(* IEC 61131-3 sources: ArfBotOS/Codesys/Scripts/st, 4 files *)

(* ---- _00_Main_decl.st ---- *)
PROGRAM _00_Main
VAR
	//
    TaskInfo : POINTER TO CmpIecTask.Task_Info2;
    TaskHandle: CmpIecTask.RTS_IEC_HANDLE;
    Result: CmpIecTask.RTS_IEC_RESULT;

	// group handler for all motion fbs
	GroupHandler: FB_GroupHandler;

	// tuning
	MoveDistance: LREAL := 5.0;
	MoveRelative: ARRAY[0..5] OF MC_MoveRelative;
	EstimateDeadTime: ARRAY[0..5] OF SMC_EstimateDeadTime;
	TuneStart: ARRAY[0..5] OF BOOL;
	TraceStart: ARRAY[0..5] OF BOOL;
	TraceStop: ARRAY[0..5] OF BOOL;
	SetTuningMoveValues: BOOL:=TRUE;
	fCycleTimeMs: LREAL; (* MainTask / SoftMotion bus cycle, ms *)
	fMeasuredLagMs: ARRAY[0..5] OF LREAL;
	fEstimatedDeadTimeRaw: ARRAY[0..5] OF LREAL; (* unclamped SMC_EstimateDeadTime median *)
	fSuggestedDeadTime: ARRAY[0..5] OF LREAL; (* D in MainTask cycles, clamped to (0, 20] *)
	nDeadTimeSamples: ARRAY[0..5] OF INT;
	bDeadTimeSuggested: ARRAY[0..5] OF BOOL;
	UseSuggestedD: ARRAY[0..5] OF BOOL;
	sDeadTimeHelp: ARRAY[0..5] OF STRING(255);

	// homing
	ProcessHome: FB_HomingProcessor;
	HomingStatusText: STRING(255);

	// jogging
	ProcessJog: FB_JogProcessor;
	JogStatusText: STRING(255);
	ButtonTextIndex: INT:=0;

	// cnc
	VisuStruct3DControl_J: VisuStruct3DControl;
	TrackPosition: PositionTracker;

	// program processor
	ProcessPrograms: FB_ProgramProcessor;
	ProcessCommand_ActiveProgram: UINT := 0;
	ActiveCommandDetails: STRING(255):='';

	// controller
	Controller: FB_Controller;

	//
	EnableRtrig: R_TRIG;
	EnableFtrig: F_TRIG;
	_i, _j, _k: INT;
	BuildTests: BOOL:=FALSE;
	FirstScan: BOOL:=TRUE;

END_VAR

(* ---- _M_Tuning_decl.st ---- *)
METHOD PRIVATE _M_Tuning : BOOL
VAR_INPUT
END_VAR
VAR_STAT
	_MoveDelayTimer: ARRAY[0..5] OF TON;
	_TraceStartFtrig: ARRAY[0..5] OF F_TRIG;
	_MoveBusyFtrig: ARRAY[0..5] OF F_TRIG;
	_MoveBusyRtrig: ARRAY[0..5] OF R_TRIG;
	_MoveDelayTime: INT:=10; // ms
	_eDtState: ARRAY[0..5] OF INT; (* 0 idle, 1 wait cruise, 2 sampling, 3 done *)
	_bEstEnable: ARRAY[0..5] OF BOOL;
	_bDtFinish: ARRAY[0..5] OF BOOL;
	_aDtSample: ARRAY[0..5, 0..63] OF LREAL;
	_nSamples: ARRAY[0..5] OF INT;
	_fSetVel: LREAL;
	_fCruiseVel: LREAL;
	_fMedian: LREAL;
	_fSwap: LREAL;
	_fDtMin: LREAL := 0.1; (* SoftMotion rejects D = 0 *)
	_fDtMax: LREAL := 20.0; (* PosControl delay-buffer limit *)
	_fCruiseRatio: LREAL := 0.9;
	_nSampleMax: INT := 64;
	_i, _j, _k: INT;
END_VAR

(* ---- _M_Tuning_impl.st ---- *)
// MainTask interval is the SoftMotion bus cycle that D is counted in.
// TaskInfo.dwInterval is microseconds (simulation writes 1000).
IF GVL.dwMainInterval > 0 THEN
	fCycleTimeMs := DWORD_TO_LREAL(GVL.dwMainInterval) / 1000.0;
ELSE
	fCycleTimeMs := 1.0;
END_IF

IF FirstScan THEN
	FOR _i:=0 TO 5 BY 1 DO
		sDeadTimeHelp[_i] := 'SMC_EstimateDeadTime: START TUNE at Kp=0. Suggested D is the median of constant-velocity samples.';
	END_FOR
END_IF

// initial values
IF SetTuningMoveValues AND_THEN PersistentVars.Flags[GVL.INIT_DRV_IDX].Value THEN
	SetTuningMoveValues := FALSE;

	MoveRelative[0].Velocity := IoConfig_Globals.J1.fSWMaxVelocity;
	MoveRelative[0].Acceleration := IoConfig_Globals.J1.fSWMaxAcceleration;
	MoveRelative[0].Deceleration := IoConfig_Globals.J1.fSWMaxDeceleration;
	MoveRelative[0].Jerk := IoConfig_Globals.J1.fSWMaxJerk;
	MoveRelative[0].Distance := MoveDistance;

	MoveRelative[1].Velocity := IoConfig_Globals.J2.fSWMaxVelocity;
	MoveRelative[1].Acceleration := IoConfig_Globals.J2.fSWMaxAcceleration;
	MoveRelative[1].Deceleration := IoConfig_Globals.J2.fSWMaxDeceleration;
	MoveRelative[1].Jerk := IoConfig_Globals.J2.fSWMaxJerk;
	MoveRelative[1].Distance := MoveDistance;

	MoveRelative[2].Velocity := IoConfig_Globals.J3.fSWMaxVelocity;
	MoveRelative[2].Acceleration := IoConfig_Globals.J3.fSWMaxAcceleration;
	MoveRelative[2].Deceleration := IoConfig_Globals.J3.fSWMaxDeceleration;
	MoveRelative[2].Jerk := IoConfig_Globals.J3.fSWMaxJerk;
	MoveRelative[2].Distance := MoveDistance;

	MoveRelative[3].Velocity := IoConfig_Globals.J4.fSWMaxVelocity;
	MoveRelative[3].Acceleration := IoConfig_Globals.J4.fSWMaxAcceleration;
	MoveRelative[3].Deceleration := IoConfig_Globals.J4.fSWMaxDeceleration;
	MoveRelative[3].Jerk := IoConfig_Globals.J4.fSWMaxJerk;
	MoveRelative[3].Distance := MoveDistance;

	MoveRelative[4].Velocity := IoConfig_Globals.J5.fSWMaxVelocity;
	MoveRelative[4].Acceleration := IoConfig_Globals.J5.fSWMaxAcceleration;
	MoveRelative[4].Deceleration := IoConfig_Globals.J5.fSWMaxDeceleration;
	MoveRelative[4].Jerk := IoConfig_Globals.J5.fSWMaxJerk;
	MoveRelative[4].Distance := MoveDistance;

	MoveRelative[5].Velocity := IoConfig_Globals.J6.fSWMaxVelocity;
	MoveRelative[5].Acceleration := IoConfig_Globals.J6.fSWMaxAcceleration;
	MoveRelative[5].Deceleration := IoConfig_Globals.J6.fSWMaxDeceleration;
	MoveRelative[5].Jerk := IoConfig_Globals.J6.fSWMaxJerk;
	MoveRelative[5].Distance := MoveDistance;
END_IF

// trace activation
FOR _i:=0 TO 5 BY 1 DO

	IF TuneStart[_i] THEN
		TuneStart[_i] := FALSE;
		TraceStart[_i] := TRUE; // trace will handshake this bit low
		GroupHandler.M_EnableGroup();
		bDeadTimeSuggested[_i] := FALSE;
		fMeasuredLagMs[_i] := 0.0;
		fEstimatedDeadTimeRaw[_i] := 0.0;
		fSuggestedDeadTime[_i] := 0.0;
		nDeadTimeSamples[_i] := 0;
		_eDtState[_i] := 0;
		_bEstEnable[_i] := FALSE;
		_bDtFinish[_i] := FALSE;
		_nSamples[_i] := 0;
		sDeadTimeHelp[_i] := 'SMC_EstimateDeadTime: waiting for constant velocity. Kp=0 gives the cleanest estimate.';
	END_IF

	// copy a valid suggestion into the DeadTime spin; WRITE PARAMETERS still applies it
	IF UseSuggestedD[_i] THEN
		UseSuggestedD[_i] := FALSE;
		IF bDeadTimeSuggested[_i] THEN
			PersistentVars.PositionControllers[_i].fDeadTime := fSuggestedDeadTime[_i];
			sDeadTimeHelp[_i] := 'Copied suggested D into DeadTime. Press WRITE PARAMETERS to apply.';
		ELSE
			sDeadTimeHelp[_i] := 'No suggested D yet. Press START TUNE first.';
		END_IF
	END_IF

	// TraceStart will clear after handshake. this means the trace has started collecting samples
	// start the move delay timer to capture samples before the move
	_TraceStartFtrig[_i](CLK:=TraceStart[_i]);
	IF _TraceStartFtrig[_i].Q THEN
		_MoveDelayTimer[_i].IN:=TRUE;
	END_IF

	// once the move delay expires, start the move
	_MoveDelayTimer[_i](PT:=INT_TO_TIME(_MoveDelayTime));
	IF _MoveDelayTimer[_i].Q THEN
		_MoveDelayTimer[_i].IN:=FALSE;
		MoveRelative[_i].Execute := TRUE;
	END_IF

	_MoveBusyFtrig[_i](CLK:=MoveRelative[_i].Busy);
	IF _MoveBusyFtrig[_i].Q THEN
		MoveRelative[_i].Execute := FALSE;
		MoveRelative[_i].Distance := MoveRelative[_i].Distance * -1.0; // reverse direction
		_bEstEnable[_i] := FALSE;
		IF _eDtState[_i] = 2 THEN
			_bDtFinish[_i] := TRUE;
		ELSIF _eDtState[_i] = 1 THEN
			_eDtState[_i] := 0;
			sDeadTimeHelp[_i] := 'Move ended before constant velocity. Increase MoveDistance or reduce acceleration.';
		END_IF
	END_IF

	CASE _i OF
		0: _fSetVel := IoConfig_Globals.J1.fSetVelocity;
		1: _fSetVel := IoConfig_Globals.J2.fSetVelocity;
		2: _fSetVel := IoConfig_Globals.J3.fSetVelocity;
		3: _fSetVel := IoConfig_Globals.J4.fSetVelocity;
		4: _fSetVel := IoConfig_Globals.J5.fSetVelocity;
		5: _fSetVel := IoConfig_Globals.J6.fSetVelocity;
	END_CASE

	_MoveBusyRtrig[_i](CLK:=MoveRelative[_i].Busy);
	IF _MoveBusyRtrig[_i].Q THEN
		_nSamples[_i] := 0;
		nDeadTimeSamples[_i] := 0;
		_bDtFinish[_i] := FALSE;
		_eDtState[_i] := 1;
	END_IF

	_fCruiseVel := MoveRelative[_i].Velocity * _fCruiseRatio;
	IF _eDtState[_i] = 1 THEN
		IF ABS(_fSetVel) >= _fCruiseVel THEN
			_bEstEnable[_i] := TRUE;
			_eDtState[_i] := 2;
			sDeadTimeHelp[_i] := 'SMC_EstimateDeadTime: sampling at constant velocity...';
		END_IF
	END_IF

	IF _eDtState[_i] = 2 THEN
		IF _bEstEnable[_i] AND EstimateDeadTime[_i].Valid AND (_nSamples[_i] < _nSampleMax) THEN
			_aDtSample[_i, _nSamples[_i]] := ABS(EstimateDeadTime[_i].DeadTimeCycles);
			_nSamples[_i] := _nSamples[_i] + 1;
			nDeadTimeSamples[_i] := _nSamples[_i];
			IF _nSamples[_i] >= _nSampleMax THEN
				_bDtFinish[_i] := TRUE;
			END_IF
		END_IF
	END_IF

	IF _bDtFinish[_i] THEN
		_bDtFinish[_i] := FALSE;
		_bEstEnable[_i] := FALSE;
		_eDtState[_i] := 3;
		IF _nSamples[_i] < 1 THEN
			_eDtState[_i] := 0;
			sDeadTimeHelp[_i] := 'SMC_EstimateDeadTime never went Valid. Check enable and that the axis reached cruise.';
		ELSE
			// median of collected DeadTimeCycles
			FOR _j:=0 TO (_nSamples[_i] - 2) BY 1 DO
				FOR _k:=(_j + 1) TO (_nSamples[_i] - 1) BY 1 DO
					IF _aDtSample[_i, _k] < _aDtSample[_i, _j] THEN
						_fSwap := _aDtSample[_i, _j];
						_aDtSample[_i, _j] := _aDtSample[_i, _k];
						_aDtSample[_i, _k] := _fSwap;
					END_IF
				END_FOR
			END_FOR
			_fMedian := ABS(_aDtSample[_i, _nSamples[_i] / 2]);
			fEstimatedDeadTimeRaw[_i] := _fMedian;
			fMeasuredLagMs[_i] := _fMedian * fCycleTimeMs;
			IF _fMedian < _fDtMin THEN
				fSuggestedDeadTime[_i] := _fDtMin;
			ELSIF _fMedian > _fDtMax THEN
				fSuggestedDeadTime[_i] := _fDtMax;
			ELSE
				fSuggestedDeadTime[_i] := _fMedian;
			END_IF
			bDeadTimeSuggested[_i] := TRUE;
			sDeadTimeHelp[_i] := 'SMC_EstimateDeadTime median ';
			sDeadTimeHelp[_i] := CONCAT(sDeadTimeHelp[_i], TO_STRING(fEstimatedDeadTimeRaw[_i]));
			sDeadTimeHelp[_i] := CONCAT(sDeadTimeHelp[_i], ' cycles (');
			sDeadTimeHelp[_i] := CONCAT(sDeadTimeHelp[_i], TO_STRING(fMeasuredLagMs[_i]));
			sDeadTimeHelp[_i] := CONCAT(sDeadTimeHelp[_i], ' ms, n=');
			sDeadTimeHelp[_i] := CONCAT(sDeadTimeHelp[_i], INT_TO_STRING(_nSamples[_i]));
			IF fEstimatedDeadTimeRaw[_i] > _fDtMax THEN
				sDeadTimeHelp[_i] := CONCAT(sDeadTimeHelp[_i], '). Clamped to D 20 (PosControl max). WRITE PARAMETERS to apply.');
			ELSE
				sDeadTimeHelp[_i] := CONCAT(sDeadTimeHelp[_i], '). Suggested D ');
				sDeadTimeHelp[_i] := CONCAT(sDeadTimeHelp[_i], TO_STRING(fSuggestedDeadTime[_i]));
				sDeadTimeHelp[_i] := CONCAT(sDeadTimeHelp[_i], '. WRITE PARAMETERS to apply.');
			END_IF
		END_IF
	END_IF

END_FOR

// official SoftMotion estimator: enable only while at constant velocity
EstimateDeadTime[0](Axis:= IoConfig_Globals.J1, Enable:= _bEstEnable[0]);
EstimateDeadTime[1](Axis:= IoConfig_Globals.J2, Enable:= _bEstEnable[1]);
EstimateDeadTime[2](Axis:= IoConfig_Globals.J3, Enable:= _bEstEnable[2]);
EstimateDeadTime[3](Axis:= IoConfig_Globals.J4, Enable:= _bEstEnable[3]);
EstimateDeadTime[4](Axis:= IoConfig_Globals.J5, Enable:= _bEstEnable[4]);
EstimateDeadTime[5](Axis:= IoConfig_Globals.J6, Enable:= _bEstEnable[5]);

// move relative
MoveRelative[0](
	Axis:= IoConfig_Globals.J1,
	Execute:= ,
	Distance:= ,
	Velocity:= ,
	Acceleration:= ,
	Deceleration:= ,
	Jerk:= ,
	BufferMode:= ,
	Done=> ,
	Busy=> ,
	Active=> ,
	CommandAborted=> ,
	Error=> ,
	ErrorID=> );
MoveRelative[1](
	Axis:= IoConfig_Globals.J2,
	Execute:= ,
	Distance:= ,
	Velocity:= ,
	Acceleration:= ,
	Deceleration:= ,
	Jerk:= ,
	BufferMode:= ,
	Done=> ,
	Busy=> ,
	Active=> ,
	CommandAborted=> ,
	Error=> ,
	ErrorID=> );
MoveRelative[2](
	Axis:= IoConfig_Globals.J3,
	Execute:= ,
	Distance:= ,
	Velocity:= ,
	Acceleration:= ,
	Deceleration:= ,
	Jerk:= ,
	BufferMode:= ,
	Done=> ,
	Busy=> ,
	Active=> ,
	CommandAborted=> ,
	Error=> ,
	ErrorID=> );
MoveRelative[3](
	Axis:= IoConfig_Globals.J4,
	Execute:= ,
	Distance:= ,
	Velocity:= ,
	Acceleration:= ,
	Deceleration:= ,
	Jerk:= ,
	BufferMode:= ,
	Done=> ,
	Busy=> ,
	Active=> ,
	CommandAborted=> ,
	Error=> ,
	ErrorID=> );
MoveRelative[4](
	Axis:= IoConfig_Globals.J5,
	Execute:= ,
	Distance:= ,
	Velocity:= ,
	Acceleration:= ,
	Deceleration:= ,
	Jerk:= ,
	BufferMode:= ,
	Done=> ,
	Busy=> ,
	Active=> ,
	CommandAborted=> ,
	Error=> ,
	ErrorID=> );
MoveRelative[5](
	Axis:= IoConfig_Globals.J6,
	Execute:= ,
	Distance:= ,
	Velocity:= ,
	Acceleration:= ,
	Deceleration:= ,
	Jerk:= ,
	BufferMode:= ,
	Done=> ,
	Busy=> ,
	Active=> ,
	CommandAborted=> ,
	Error=> ,
	ErrorID=> );

(* ---- M_BuildTests_impl.st ---- *)
// taught positions referenced by factory programs
PersistentVars.StoredPositions[40].Position.X := -76.81;
PersistentVars.StoredPositions[40].Position.Y := 1.2;
PersistentVars.StoredPositions[40].Position.Z := -24.93;
PersistentVars.StoredPositions[40].Position.A := -4.74;
PersistentVars.StoredPositions[40].Position.B := 62.93;
PersistentVars.StoredPositions[40].Position.C := 24.21;
PersistentVars.StoredPositions[41].Comment := 'Euler Angle Tool Place Position MCS';
PersistentVars.StoredPositions[41].Position.X := 44.39;
PersistentVars.StoredPositions[41].Position.Y := -285.95;
PersistentVars.StoredPositions[41].Position.Z := 310.15;
PersistentVars.StoredPositions[41].Position.A := 96.6;
PersistentVars.StoredPositions[41].Position.B := 177.75;
PersistentVars.StoredPositions[41].Position.C := -174.21;
PersistentVars.StoredPositions[42].Comment := 'Euler Angle Tool Pick Position MCS';
PersistentVars.StoredPositions[42].Position.X := 43.97;
PersistentVars.StoredPositions[42].Position.Y := -280.38;
PersistentVars.StoredPositions[42].Position.Z := 215.24;
PersistentVars.StoredPositions[42].Position.A := 96.61;
PersistentVars.StoredPositions[42].Position.B := 177.75;
PersistentVars.StoredPositions[42].Position.C := -174.22;

//
FOR _i := GVL.PROG_CMDS_ARR_BEG TO GVL.PROG_CMDS_ARR_END BY 1 DO
	PersistentVars.Programs[0].Commands[_i].CommandType := DUT_CommandType.Disabled;
	PersistentVars.Programs[0].Commands[_i].CommandString := '';
	PersistentVars.Programs[0].Commands[_i].CommandComment := '';
END_FOR
PersistentVars.Programs[0].ProgramName := 'Pick and Place Euler Angle Tool';
PersistentVars.Programs[0].Commands[0].CommandType := DUT_CommandType.MoveCommand;
PersistentVars.Programs[0].Commands[0].CommandString := 'DIR ABS 50.0 ACS VAR STO 35 ';
PersistentVars.Programs[0].Commands[0].CommandComment := 'take on a pose';
PersistentVars.Programs[0].Commands[1].CommandType := DUT_CommandType.VarSetCommand;
PersistentVars.Programs[0].Commands[1].CommandString := 'STO 46 E 0.0 E 0.0 E 0.0 E 0.0 E 0.0 E 0.0 ';
PersistentVars.Programs[0].Commands[1].CommandComment := 'Rotate TCP according to ZYZ convention';
PersistentVars.Programs[0].Commands[3].CommandType := DUT_CommandType.LogicCommand;
PersistentVars.Programs[0].Commands[3].CommandString := 'IF REGISTER 40 EQU 0 THEN JUMP 5 ELSE JUMP 12 ';
PersistentVars.Programs[0].Commands[3].CommandComment := 'determine if pick or place';
PersistentVars.Programs[0].Commands[5].CommandType := DUT_CommandType.MoveCommand;
PersistentVars.Programs[0].Commands[5].CommandString := 'DIR ABS 50.0 MCS VAR STO 42 ';
PersistentVars.Programs[0].Commands[5].CommandComment := 'go to euler angle tool down position';
PersistentVars.Programs[0].Commands[6].CommandType := DUT_CommandType.OutputCommand;
PersistentVars.Programs[0].Commands[6].CommandString := 'DIG 0 1.0 ';
PersistentVars.Programs[0].Commands[6].CommandComment := 'open gripper';
PersistentVars.Programs[0].Commands[7].CommandType := DUT_CommandType.MoveCommand;
PersistentVars.Programs[0].Commands[7].CommandString := 'LIN REL 20.0 TCS LIT 0.0 0.0 25.0 0.0 0.0 0.0 ';
PersistentVars.Programs[0].Commands[7].CommandComment := 'move onto euler angle tool';
PersistentVars.Programs[0].Commands[8].CommandType := DUT_CommandType.OutputCommand;
PersistentVars.Programs[0].Commands[8].CommandString := 'DIG 0 0.0 ';
PersistentVars.Programs[0].Commands[8].CommandComment := 'close gripper';
PersistentVars.Programs[0].Commands[9].CommandType := DUT_CommandType.MoveCommand;
PersistentVars.Programs[0].Commands[9].CommandString := 'LIN REL 20.0 TCS LIT 0.0 0.0 -120.0 0.0 0.0 0.0 ';
PersistentVars.Programs[0].Commands[9].CommandComment := 'pull out tool';
PersistentVars.Programs[0].Commands[10].CommandType := DUT_CommandType.LogicCommand;
PersistentVars.Programs[0].Commands[10].CommandString := 'IF PASS THEN JUMP 16 ';
PersistentVars.Programs[0].Commands[12].CommandType := DUT_CommandType.MoveCommand;
PersistentVars.Programs[0].Commands[12].CommandString := 'DIR ABS 50.0 MCS VAR STO 41 ';
PersistentVars.Programs[0].Commands[12].CommandComment := 'go to euler angle tool up position';
PersistentVars.Programs[0].Commands[13].CommandType := DUT_CommandType.MoveCommand;
PersistentVars.Programs[0].Commands[13].CommandString := 'LIN REL 20.0 TCS LIT 0.0 0.0 120.0 0.0 0.0 0.0 ';
PersistentVars.Programs[0].Commands[13].CommandComment := 'push tool in';
PersistentVars.Programs[0].Commands[14].CommandType := DUT_CommandType.OutputCommand;
PersistentVars.Programs[0].Commands[14].CommandString := 'DIG 0 1.0 ';
PersistentVars.Programs[0].Commands[14].CommandComment := 'open gripper';
PersistentVars.Programs[0].Commands[15].CommandType := DUT_CommandType.MoveCommand;
PersistentVars.Programs[0].Commands[15].CommandString := 'LIN REL 20.0 TCS LIT 0.0 0.0 -25.0 0.0 0.0 0.0 ';
PersistentVars.Programs[0].Commands[15].CommandComment := 'move away from euler angle tool';

//
FOR _i := GVL.PROG_CMDS_ARR_BEG TO GVL.PROG_CMDS_ARR_END BY 1 DO
	PersistentVars.Programs[1].Commands[_i].CommandType := DUT_CommandType.Disabled;
	PersistentVars.Programs[1].Commands[_i].CommandString := '';
	PersistentVars.Programs[1].Commands[_i].CommandComment := '';
END_FOR
PersistentVars.Programs[1].ProgramName := 'Vision Pick and Place';
PersistentVars.Programs[1].Commands[0].CommandType := DUT_CommandType.VarSetCommand;
PersistentVars.Programs[1].Commands[0].CommandString := 'STO 46 E 0.0 E 0.0 E 0.0 E 0.0 E 0.0 E 90.0 ';
PersistentVars.Programs[1].Commands[0].CommandComment := 'Rotate TCP according to ZYZ convention';
PersistentVars.Programs[1].Commands[1].CommandType := DUT_CommandType.MoveCommand;
PersistentVars.Programs[1].Commands[1].CommandString := 'DIR ABS 60.0 ACS VAR STO 40 ';
PersistentVars.Programs[1].Commands[1].CommandComment := 'Take a pose';
PersistentVars.Programs[1].Commands[2].CommandType := DUT_CommandType.VisionCommand;
PersistentVars.Programs[1].Commands[2].CommandString := 'LOC 640 400 15 1 0.0 0.6 180.0 0 Pen.jpg FastTemplateMatching.py ';
PersistentVars.Programs[1].Commands[2].CommandComment := 'Find the object and store the result';
PersistentVars.Programs[1].Commands[3].CommandType := DUT_CommandType.VarSetCommand;
PersistentVars.Programs[1].Commands[3].CommandString := 'VIS 0 M -1.0 M -1.0 E -20.0 M -1.0 N 0.0 N 0.0 ';
PersistentVars.Programs[1].Commands[3].CommandComment := 'Rotate x and y to line up with TCP';
PersistentVars.Programs[1].Commands[4].CommandType := DUT_CommandType.MoveCommand;
PersistentVars.Programs[1].Commands[4].CommandString := 'DIR ABS 50.0 PC1 VAR VIS 0 ';
PersistentVars.Programs[1].Commands[4].CommandComment := 'Move over the object';
PersistentVars.Programs[1].Commands[5].CommandType := DUT_CommandType.OutputCommand;
PersistentVars.Programs[1].Commands[5].CommandString := 'DIG 0 1.0 ';
PersistentVars.Programs[1].Commands[5].CommandComment := 'Open the Gripper';
PersistentVars.Programs[1].Commands[6].CommandType := DUT_CommandType.MoveCommand;
PersistentVars.Programs[1].Commands[6].CommandString := 'LIN REL 50.0 TCS LIT 0.0 0.0 20.0 0.0 0.0 0.0 ';
PersistentVars.Programs[1].Commands[6].CommandComment := 'Move down to the object';
PersistentVars.Programs[1].Commands[7].CommandType := DUT_CommandType.OutputCommand;
PersistentVars.Programs[1].Commands[7].CommandString := 'DIG 0 0.0 ';
PersistentVars.Programs[1].Commands[7].CommandComment := 'Close the Gripper';
PersistentVars.Programs[1].Commands[8].CommandType := DUT_CommandType.PauseCommand;
PersistentVars.Programs[1].Commands[8].CommandString := 'T#1s';
PersistentVars.Programs[1].Commands[8].CommandComment := 'Pause while the gripper closes';
PersistentVars.Programs[1].Commands[9].CommandType := DUT_CommandType.MoveCommand;
PersistentVars.Programs[1].Commands[9].CommandString := 'LIN REL 50.0 TCS LIT 0.0 0.0 -20.0 0.0 0.0 0.0 ';
PersistentVars.Programs[1].Commands[9].CommandComment := 'Pick up the object';
PersistentVars.Programs[1].Commands[10].CommandType := DUT_CommandType.MoveCommand;
PersistentVars.Programs[1].Commands[10].CommandString := 'DIR ABS 50.0 PC1 LIT 0.0 0.0 -50.0 0.0 0.0 90.0 ';
PersistentVars.Programs[1].Commands[10].CommandComment := 'Move to drop position';
PersistentVars.Programs[1].Commands[11].CommandType := DUT_CommandType.OutputCommand;
PersistentVars.Programs[1].Commands[11].CommandString := 'DIG 0 1.0 ';
PersistentVars.Programs[1].Commands[11].CommandComment := 'Open the Gripper';

//
FOR _i := GVL.PROG_CMDS_ARR_BEG TO GVL.PROG_CMDS_ARR_END BY 1 DO
	PersistentVars.Programs[2].Commands[_i].CommandType := DUT_CommandType.Disabled;
	PersistentVars.Programs[2].Commands[_i].CommandString := '';
	PersistentVars.Programs[2].Commands[_i].CommandComment := '';
END_FOR
PersistentVars.Programs[2].ProgramName := 'PCS1 Corners';
PersistentVars.Programs[2].Commands[0].CommandType := DUT_CommandType.VarSetCommand;
PersistentVars.Programs[2].Commands[0].CommandString := 'STO 46 E 0.0 E 0.0 E 0.0 E 180.0 E 180.0 E 0.0 ';
PersistentVars.Programs[2].Commands[0].CommandComment := 'Rotate TCP according to ZYZ convention';
PersistentVars.Programs[2].Commands[1].CommandType := DUT_CommandType.VarSetCommand;
PersistentVars.Programs[2].Commands[1].CommandString := 'STO 48 E 282.23 E -0066.77 E 0195.00 E 0.0 E 0.0 E -0030.00 ';
PersistentVars.Programs[2].Commands[2].CommandType := DUT_CommandType.MoveCommand;
PersistentVars.Programs[2].Commands[2].CommandString := 'DIR ABS 050 PC1 LIT 0 0 0 0 0 0';
PersistentVars.Programs[2].Commands[3].CommandType := DUT_CommandType.MoveCommand;
PersistentVars.Programs[2].Commands[3].CommandString := 'LIN REL 100 TCS LIT 0.0 200.0 0.0 0.0 0.0 0.0';
PersistentVars.Programs[2].Commands[4].CommandType := DUT_CommandType.MoveCommand;
PersistentVars.Programs[2].Commands[4].CommandString := 'LIN REL 100 TCS LIT 00125.00 00000.00 00000.00 00000.00 00000.00 00000.00';
PersistentVars.Programs[2].Commands[5].CommandType := DUT_CommandType.MoveCommand;
PersistentVars.Programs[2].Commands[5].CommandString := 'LIN REL 100 TCS LIT 00000.00 -0200.00 00000.00 00000.00 00000.00 00000.00';
PersistentVars.Programs[2].Commands[6].CommandType := DUT_CommandType.MoveCommand;
PersistentVars.Programs[2].Commands[6].CommandString := 'LIN REL 100 TCS LIT -0125.00 00000.00 00000.00 00000.00 00000.00 00000.00';
PersistentVars.Programs[2].Commands[7].CommandType := DUT_CommandType.MoveCommand;
PersistentVars.Programs[2].Commands[7].CommandString := 'DIR ABS 050 ACS LIT +00 +30 -30 +00 +30 +00';

//
FOR _i := GVL.PROG_CMDS_ARR_BEG TO GVL.PROG_CMDS_ARR_END BY 1 DO
	PersistentVars.Programs[3].Commands[_i].CommandType := DUT_CommandType.Disabled;
	PersistentVars.Programs[3].Commands[_i].CommandString := '';
	PersistentVars.Programs[3].Commands[_i].CommandComment := '';
END_FOR
PersistentVars.Programs[3].ProgramName := 'Cnc Validation';
PersistentVars.Programs[3].Commands[0].CommandType := DUT_CommandType.VarSetCommand;
PersistentVars.Programs[3].Commands[0].CommandString := 'STO 46 E 0.0 E 0.0 E 0.0 E 0.0 E 0.0 E 0.0 ';
PersistentVars.Programs[3].Commands[0].CommandComment := 'Clear TCP Offset';
PersistentVars.Programs[3].Commands[2].CommandType := DUT_CommandType.MoveCommand;
PersistentVars.Programs[3].Commands[2].CommandString := 'DIR ABS 50.0 ACS VAR STO 37 ';
PersistentVars.Programs[3].Commands[2].CommandComment := 'Move to Pose 4';
PersistentVars.Programs[3].Commands[3].CommandType := DUT_CommandType.CncCommand;
PersistentVars.Programs[3].Commands[3].CommandString := 'CNC_Cone.cnc ';
PersistentVars.Programs[3].Commands[3].CommandComment := 'Run the cnc file on disk';
PersistentVars.Programs[3].Commands[5].CommandType := DUT_CommandType.MoveCommand;
PersistentVars.Programs[3].Commands[5].CommandString := 'DIR ABS 50.0 ACS VAR STO 34 ';
PersistentVars.Programs[3].Commands[5].CommandComment := 'Move to Pose 1';
PersistentVars.Programs[3].Commands[6].CommandType := DUT_CommandType.CncCommand;
PersistentVars.Programs[3].Commands[6].CommandString := 'CNC_FromFile.cnc ';
PersistentVars.Programs[3].Commands[6].CommandComment := 'Run the cnc file on disk';

//
FOR _i := GVL.PROG_CMDS_ARR_BEG TO GVL.PROG_CMDS_ARR_END BY 1 DO
	PersistentVars.Programs[4].Commands[_i].CommandType := DUT_CommandType.Disabled;
	PersistentVars.Programs[4].Commands[_i].CommandString := '';
	PersistentVars.Programs[4].Commands[_i].CommandComment := '';
END_FOR
PersistentVars.Programs[4].ProgramName := 'Vision Validation';
PersistentVars.Programs[4].Commands[0].CommandType := DUT_CommandType.VisionCommand;
PersistentVars.Programs[4].Commands[0].CommandString := 'CAL 640 400 60 22.0 6 9 ';
PersistentVars.Programs[4].Commands[0].CommandComment := 'Calibrate using checkerboard';
PersistentVars.Programs[4].Commands[2].CommandType := DUT_CommandType.PauseCommand;
PersistentVars.Programs[4].Commands[2].CommandString := 'T#10s ';
PersistentVars.Programs[4].Commands[2].CommandComment := 'Wait 10 seconds';
PersistentVars.Programs[4].Commands[4].CommandType := DUT_CommandType.VisionCommand;
PersistentVars.Programs[4].Commands[4].CommandString := 'LOC 640 400 60 1 0.0 0.8 30.0 10 Template.jpg FastTemplateMatching.py';
PersistentVars.Programs[4].Commands[4].CommandComment := 'Find the template';

//
FOR _i := GVL.PROG_CMDS_ARR_BEG TO GVL.PROG_CMDS_ARR_END BY 1 DO
	PersistentVars.Programs[5].Commands[_i].CommandType := DUT_CommandType.Disabled;
	PersistentVars.Programs[5].Commands[_i].CommandString := '';
	PersistentVars.Programs[5].Commands[_i].CommandComment := '';
END_FOR
PersistentVars.Programs[5].ProgramName := 'VarSet Validation';
PersistentVars.Programs[5].Commands[0].CommandType := DUT_CommandType.VarSetCommand;
PersistentVars.Programs[5].Commands[0].CommandString := 'STO 1 E 6.0 E 5.0 E 4.0 E 3.0 E 2.0 E 1.0 ';
PersistentVars.Programs[5].Commands[1].CommandType := DUT_CommandType.VarSetCommand;
PersistentVars.Programs[5].Commands[1].CommandString := 'VIS 2 1 2 3 4 5 6';
PersistentVars.Programs[5].Commands[2].CommandType := DUT_CommandType.VarSetCommand;
PersistentVars.Programs[5].Commands[2].CommandString := 'FLG 3 1';

//
FOR _i := GVL.PROG_CMDS_ARR_BEG TO GVL.PROG_CMDS_ARR_END BY 1 DO
	PersistentVars.Programs[6].Commands[_i].CommandType := DUT_CommandType.Disabled;
	PersistentVars.Programs[6].Commands[_i].CommandString := '';
	PersistentVars.Programs[6].Commands[_i].CommandComment := '';
END_FOR
PersistentVars.Programs[6].ProgramName := 'Logic Validation';
PersistentVars.Programs[6].Commands[0].CommandType := DUT_CommandType.LogicCommand;
PersistentVars.Programs[6].Commands[0].CommandString := 'IF INPUT 1 EQU 1 THEN OUTPUT 1 1 ELSE OUTPUT 1 0';
PersistentVars.Programs[6].Commands[1].CommandType := DUT_CommandType.LogicCommand;
PersistentVars.Programs[6].Commands[1].CommandString := 'IF INPUT 1 EQU 1 THEN CNTUP 1 ELSE CNTUP 2';
PersistentVars.Programs[6].Commands[2].CommandType := DUT_CommandType.LogicCommand;
PersistentVars.Programs[6].Commands[2].CommandString := 'IF COUNTER 2 GRE 10 THEN NOP ELSE JUMP 0';

//
FOR _i := GVL.PROG_CMDS_ARR_BEG TO GVL.PROG_CMDS_ARR_END BY 1 DO
	PersistentVars.Programs[7].Commands[_i].CommandType := DUT_CommandType.Disabled;
	PersistentVars.Programs[7].Commands[_i].CommandString := '';
	PersistentVars.Programs[7].Commands[_i].CommandComment := '';
END_FOR
PersistentVars.Programs[7].ProgramName := 'Euler Angles Demo';
PersistentVars.Programs[7].Commands[0].CommandType := DUT_CommandType.LogicCommand;
PersistentVars.Programs[7].Commands[0].CommandString := 'IF PASS THEN REGISTER 40 0 ';
PersistentVars.Programs[7].Commands[0].CommandComment := 'Set pick/place register to pick tool';
PersistentVars.Programs[7].Commands[1].CommandType := DUT_CommandType.LogicCommand;
PersistentVars.Programs[7].Commands[1].CommandString := 'IF PASS THEN CALL 0 ';
PersistentVars.Programs[7].Commands[1].CommandComment := 'Call pick and place program';
PersistentVars.Programs[7].Commands[3].CommandType := DUT_CommandType.LogicCommand;
PersistentVars.Programs[7].Commands[3].CommandString := 'IF COUNTER 7 EQU 0 THEN NOP ELSE JUMP 7 ';
PersistentVars.Programs[7].Commands[3].CommandComment := 'apply or jump over';
PersistentVars.Programs[7].Commands[4].CommandType := DUT_CommandType.VarSetCommand;
PersistentVars.Programs[7].Commands[4].CommandString := 'STO 46 E 0.0 E 0.0 E 70.0 E 0.0 E 0.0 E 0.0 ';
PersistentVars.Programs[7].Commands[4].CommandComment := 'offset TCP Z';
PersistentVars.Programs[7].Commands[5].CommandType := DUT_CommandType.LogicCommand;
PersistentVars.Programs[7].Commands[5].CommandString := 'IF PASS THEN JUMP 19 ';
PersistentVars.Programs[7].Commands[5].CommandComment := 'go to move commands';
PersistentVars.Programs[7].Commands[7].CommandType := DUT_CommandType.LogicCommand;
PersistentVars.Programs[7].Commands[7].CommandString := 'IF COUNTER 7 EQU 1 THEN NOP ELSE JUMP 11 ';
PersistentVars.Programs[7].Commands[7].CommandComment := 'apply or jump over';
PersistentVars.Programs[7].Commands[8].CommandType := DUT_CommandType.VarSetCommand;
PersistentVars.Programs[7].Commands[8].CommandString := 'STO 46 E 0.0 E 0.0 E 170.0 E 0.0 E 0.0 E 0.0 ';
PersistentVars.Programs[7].Commands[8].CommandComment := 'offset TCP Z';
PersistentVars.Programs[7].Commands[9].CommandType := DUT_CommandType.LogicCommand;
PersistentVars.Programs[7].Commands[9].CommandString := 'IF PASS THEN JUMP 19 ';
PersistentVars.Programs[7].Commands[9].CommandComment := 'go to move commands';
PersistentVars.Programs[7].Commands[11].CommandType := DUT_CommandType.LogicCommand;
PersistentVars.Programs[7].Commands[11].CommandString := 'IF COUNTER 7 EQU 2 THEN NOP ELSE JUMP 15 ';
PersistentVars.Programs[7].Commands[11].CommandComment := 'apply or jump over';
PersistentVars.Programs[7].Commands[12].CommandType := DUT_CommandType.VarSetCommand;
PersistentVars.Programs[7].Commands[12].CommandString := 'STO 46 E 0.0 E -100.0 E 70.0 E 0.0 E 0.0 E 0.0 ';
PersistentVars.Programs[7].Commands[12].CommandComment := 'offset TCP X and Y';
PersistentVars.Programs[7].Commands[13].CommandType := DUT_CommandType.LogicCommand;
PersistentVars.Programs[7].Commands[13].CommandString := 'IF PASS THEN JUMP 19 ';
PersistentVars.Programs[7].Commands[13].CommandComment := 'go to move commands';
PersistentVars.Programs[7].Commands[15].CommandType := DUT_CommandType.LogicCommand;
PersistentVars.Programs[7].Commands[15].CommandString := 'IF COUNTER 7 EQU 3 THEN NOP ELSE JUMP 29 ';
PersistentVars.Programs[7].Commands[15].CommandComment := 'apply or jump over';
PersistentVars.Programs[7].Commands[16].CommandType := DUT_CommandType.VarSetCommand;
PersistentVars.Programs[7].Commands[16].CommandString := 'STO 46 E 100.0 E 0.0 E 70.0 E 0.0 E 0.0 E 0.0 ';
PersistentVars.Programs[7].Commands[16].CommandComment := 'offset TCP X and Z';
PersistentVars.Programs[7].Commands[17].CommandType := DUT_CommandType.LogicCommand;
PersistentVars.Programs[7].Commands[17].CommandString := 'IF PASS THEN JUMP 19 ';
PersistentVars.Programs[7].Commands[17].CommandComment := 'go to move commands';
PersistentVars.Programs[7].Commands[19].CommandType := DUT_CommandType.MoveCommand;
PersistentVars.Programs[7].Commands[19].CommandString := 'DIR ABS 50.0 ACS VAR STO 35 ';
PersistentVars.Programs[7].Commands[19].CommandComment := 'take on a pose';
PersistentVars.Programs[7].Commands[20].CommandType := DUT_CommandType.MoveCommand;
PersistentVars.Programs[7].Commands[20].CommandString := 'LIN ABS 70.0 TCS LIT 0.0 0.0 0.0 0.0 0.0 -45.0 ';
PersistentVars.Programs[7].Commands[20].CommandComment := 'rotate TCP Z with ZYZ convention';
PersistentVars.Programs[7].Commands[21].CommandType := DUT_CommandType.MoveCommand;
PersistentVars.Programs[7].Commands[21].CommandString := 'LIN ABS 70.0 TCS LIT 0.0 0.0 0.0 0.0 -30.0 0.0 ';
PersistentVars.Programs[7].Commands[21].CommandComment := 'rotate around TCP Y with ZYZ convention';
PersistentVars.Programs[7].Commands[22].CommandType := DUT_CommandType.MoveCommand;
PersistentVars.Programs[7].Commands[22].CommandString := 'LIN ABS 70.0 TCS LIT 0.0 0.0 0.0 90.0 30.0 -90.0 ';
PersistentVars.Programs[7].Commands[22].CommandComment := 'rotate around TCP X with ZYZ convention';
PersistentVars.Programs[7].Commands[23].CommandType := DUT_CommandType.MoveCommand;
PersistentVars.Programs[7].Commands[23].CommandString := 'LIN ABS 70.0 TCS LIT 0.0 0.0 0.0 90.0 -30.0 -90.0 ';
PersistentVars.Programs[7].Commands[23].CommandComment := 'rotate around TCP X with ZYZ convention';
PersistentVars.Programs[7].Commands[24].CommandType := DUT_CommandType.MoveCommand;
PersistentVars.Programs[7].Commands[24].CommandString := 'LIN ABS 70.0 TCS LIT 0.0 0.0 0.0 0.0 30.0 0.0 ';
PersistentVars.Programs[7].Commands[24].CommandComment := 'rotate around TCP Y with ZYZ convention';
PersistentVars.Programs[7].Commands[25].CommandType := DUT_CommandType.MoveCommand;
PersistentVars.Programs[7].Commands[25].CommandString := 'DIR ABS 70.0 ACS VAR STO 35 ';
PersistentVars.Programs[7].Commands[25].CommandComment := 'take on a pose';
PersistentVars.Programs[7].Commands[27].CommandType := DUT_CommandType.LogicCommand;
PersistentVars.Programs[7].Commands[27].CommandString := 'IF PASS THEN CNTUP 7 ';
PersistentVars.Programs[7].Commands[27].CommandComment := 'count up counter';
PersistentVars.Programs[7].Commands[28].CommandType := DUT_CommandType.LogicCommand;
PersistentVars.Programs[7].Commands[28].CommandString := 'IF PASS THEN JUMP 3 ';
PersistentVars.Programs[7].Commands[28].CommandComment := 'go back to start';
PersistentVars.Programs[7].Commands[29].CommandType := DUT_CommandType.LogicCommand;
PersistentVars.Programs[7].Commands[29].CommandString := 'IF PASS THEN CNTRST 7 ';
PersistentVars.Programs[7].Commands[29].CommandComment := 'reset counter back to 0';
PersistentVars.Programs[7].Commands[31].CommandType := DUT_CommandType.LogicCommand;
PersistentVars.Programs[7].Commands[31].CommandString := 'IF PASS THEN REGISTER 40 1 ';
PersistentVars.Programs[7].Commands[31].CommandComment := 'Set pick/place register to place tool';
PersistentVars.Programs[7].Commands[32].CommandType := DUT_CommandType.LogicCommand;
PersistentVars.Programs[7].Commands[32].CommandString := 'IF PASS THEN CALL 0 ';
PersistentVars.Programs[7].Commands[32].CommandComment := 'Call pick and place program';

//
FOR _i := GVL.PROG_CMDS_ARR_BEG TO GVL.PROG_CMDS_ARR_END BY 1 DO
	PersistentVars.Programs[9].Commands[_i].CommandType := DUT_CommandType.Disabled;
	PersistentVars.Programs[9].Commands[_i].CommandString := '';
	PersistentVars.Programs[9].Commands[_i].CommandComment := '';
END_FOR
PersistentVars.Programs[9].ProgramName := 'Vision PCS1 Test';
PersistentVars.Programs[9].Commands[0].CommandType := DUT_CommandType.MoveCommand;
PersistentVars.Programs[9].Commands[0].CommandString := 'DIR ABS 75.0 ACS VAR STO 35 ';
PersistentVars.Programs[9].Commands[0].CommandComment := 'Move to Pose 2';
PersistentVars.Programs[9].Commands[2].CommandType := DUT_CommandType.VarSetCommand;
PersistentVars.Programs[9].Commands[2].CommandString := 'STO 48 E 241.75 E -54.39 E 203.17 E 0.0 E 181.0 E -90.0 ';
PersistentVars.Programs[9].Commands[2].CommandComment := 'Set PCS1 Offset in ZYZ';
PersistentVars.Programs[9].Commands[3].CommandType := DUT_CommandType.VarSetCommand;
PersistentVars.Programs[9].Commands[3].CommandString := 'STO 46 E 0.0 E 0.0 E 0.0 E 0.0 E 0.0 E 90.0 ';
PersistentVars.Programs[9].Commands[3].CommandComment := 'Rotate TCP in ZYZ';
PersistentVars.Programs[9].Commands[5].CommandType := DUT_CommandType.VisionCommand;
PersistentVars.Programs[9].Commands[5].CommandString := 'LOC 640 400 15 2 0.0 0.8 180.0 0 screwdriver1.jpg FastTemplateMatching.py ';
PersistentVars.Programs[9].Commands[5].CommandComment := 'Find the object and store the result';
PersistentVars.Programs[9].Commands[7].CommandType := DUT_CommandType.LogicCommand;
PersistentVars.Programs[9].Commands[7].CommandString := 'IF REGISTER 0 EQU 0 THEN JUMP 14 ELSE NOP ';
PersistentVars.Programs[9].Commands[7].CommandComment := 'If parts count = 0 jump to end';
PersistentVars.Programs[9].Commands[9].CommandType := DUT_CommandType.MoveCommand;
PersistentVars.Programs[9].Commands[9].CommandString := 'DIR ABS 50.0 PC1 VAR VIS 0 ';
PersistentVars.Programs[9].Commands[9].CommandComment := 'Move over the object';
PersistentVars.Programs[9].Commands[10].CommandType := DUT_CommandType.PauseCommand;
PersistentVars.Programs[9].Commands[10].CommandString := 'T#3s ';
PersistentVars.Programs[9].Commands[12].CommandType := DUT_CommandType.LogicCommand;
PersistentVars.Programs[9].Commands[12].CommandString := 'IF REGISTER 0 GRT 1 THEN JUMP 0 ELSE NOP ';
PersistentVars.Programs[9].Commands[12].CommandComment := 'If more than 1 part go again';
PersistentVars.Programs[9].Commands[14].CommandType := DUT_CommandType.MoveCommand;
PersistentVars.Programs[9].Commands[14].CommandString := 'DIR ABS 75.0 ACS VAR STO 35 ';
PersistentVars.Programs[9].Commands[14].CommandComment := 'Move to Pose 2';

//
FOR _i := GVL.PROG_CMDS_ARR_BEG TO GVL.PROG_CMDS_ARR_END BY 1 DO
	PersistentVars.Programs[10].Commands[_i].CommandType := DUT_CommandType.Disabled;
	PersistentVars.Programs[10].Commands[_i].CommandString := '';
	PersistentVars.Programs[10].Commands[_i].CommandComment := '';
END_FOR
PersistentVars.Programs[10].ProgramName := 'Pick Glow Stick';
PersistentVars.Programs[10].Commands[0].CommandType := DUT_CommandType.LogicCommand;
PersistentVars.Programs[10].Commands[0].CommandString := 'IF REGISTER 2 EQU 0 THEN NOP ELSE JUMP 5 ';
PersistentVars.Programs[10].Commands[0].CommandComment := 'check if initialized';
PersistentVars.Programs[10].Commands[1].CommandType := DUT_CommandType.VarSetCommand;
PersistentVars.Programs[10].Commands[1].CommandString := 'STO 0 E 0.0 E 0.0 E 0.0 E 0.0 E 0.0 E 0.0 ';
PersistentVars.Programs[10].Commands[1].CommandComment := 'clear out the tcp position';
PersistentVars.Programs[10].Commands[2].CommandType := DUT_CommandType.LogicCommand;
PersistentVars.Programs[10].Commands[2].CommandString := 'IF PASS THEN CNTRST 0 ';
PersistentVars.Programs[10].Commands[2].CommandComment := 'clear column counter';
PersistentVars.Programs[10].Commands[3].CommandType := DUT_CommandType.LogicCommand;
PersistentVars.Programs[10].Commands[3].CommandString := 'IF PASS THEN CNTRST 1 ';
PersistentVars.Programs[10].Commands[3].CommandComment := 'clear row counter';
PersistentVars.Programs[10].Commands[4].CommandType := DUT_CommandType.LogicCommand;
PersistentVars.Programs[10].Commands[4].CommandString := 'IF PASS THEN REGISTER 2 1 ';
PersistentVars.Programs[10].Commands[4].CommandComment := 'mark data initialized';
PersistentVars.Programs[10].Commands[6].CommandType := DUT_CommandType.MoveCommand;
PersistentVars.Programs[10].Commands[6].CommandString := 'DIR ABS 50.0 ACS VAR STO 34 ';
PersistentVars.Programs[10].Commands[6].CommandComment := 'take on a pose';
PersistentVars.Programs[10].Commands[7].CommandType := DUT_CommandType.OutputCommand;
PersistentVars.Programs[10].Commands[7].CommandString := 'DIG 0 1.0 ';
PersistentVars.Programs[10].Commands[7].CommandComment := 'open gripper';
PersistentVars.Programs[10].Commands[8].CommandType := DUT_CommandType.MoveCommand;
PersistentVars.Programs[10].Commands[8].CommandString := 'LIN ABS 50.0 PC1 VAR STO 0 ';
PersistentVars.Programs[10].Commands[8].CommandComment := 'go to the pick position in PCS1';
PersistentVars.Programs[10].Commands[9].CommandType := DUT_CommandType.MoveCommand;
PersistentVars.Programs[10].Commands[9].CommandString := 'LIN REL 50.0 TCS LIT 0.0 0.0 10.0 0.0 0.0 0.0 ';
PersistentVars.Programs[10].Commands[9].CommandComment := 'move into glow stick';
PersistentVars.Programs[10].Commands[10].CommandType := DUT_CommandType.OutputCommand;
PersistentVars.Programs[10].Commands[10].CommandString := 'DIG 0 0.0 ';
PersistentVars.Programs[10].Commands[10].CommandComment := 'close gripper';
PersistentVars.Programs[10].Commands[11].CommandType := DUT_CommandType.MoveCommand;
PersistentVars.Programs[10].Commands[11].CommandString := 'LIN REL 50.0 TCS LIT 160.0 0.0 0.0 0.0 0.0 0.0 ';
PersistentVars.Programs[10].Commands[11].CommandComment := 'pick glow stick out of nest';
PersistentVars.Programs[10].Commands[12].CommandType := DUT_CommandType.MoveCommand;
PersistentVars.Programs[10].Commands[12].CommandString := 'LIN ABS 50.0 PC2 LIT 0.0 0.0 0.0 0.0 0.0 0.0 ';
PersistentVars.Programs[10].Commands[12].CommandComment := 'go to the home position of PCS2';
PersistentVars.Programs[10].Commands[13].CommandType := DUT_CommandType.MoveCommand;
PersistentVars.Programs[10].Commands[13].CommandString := 'LIN REL 50.0 TCS LIT 0.0 0.0 50.0 0.0 0.0 0.0 ';
PersistentVars.Programs[10].Commands[13].CommandComment := 'move into drop position';
PersistentVars.Programs[10].Commands[14].CommandType := DUT_CommandType.OutputCommand;
PersistentVars.Programs[10].Commands[14].CommandString := 'DIG 0 1.0 ';
PersistentVars.Programs[10].Commands[14].CommandComment := 'open gripper';
PersistentVars.Programs[10].Commands[15].CommandType := DUT_CommandType.MoveCommand;
PersistentVars.Programs[10].Commands[15].CommandString := 'LIN ABS 50.0 PC2 LIT 0.0 0.0 0.0 0.0 0.0 0.0 ';
PersistentVars.Programs[10].Commands[15].CommandComment := 'go to the home position of PCS2';
PersistentVars.Programs[10].Commands[17].CommandType := DUT_CommandType.LogicCommand;
PersistentVars.Programs[10].Commands[17].CommandString := 'IF COUNTER 0 LES 3 THEN CNTUP 0 ELSE JUMP 21 ';
PersistentVars.Programs[10].Commands[17].CommandComment := 'increment the column counter';
PersistentVars.Programs[10].Commands[18].CommandType := DUT_CommandType.VarSetCommand;
PersistentVars.Programs[10].Commands[18].CommandString := 'STO 0 N 0.0 A 20.0 N 0.0 N 0.0 N 0.0 N 0.0 ';
PersistentVars.Programs[10].Commands[18].CommandComment := 'add the column width';
PersistentVars.Programs[10].Commands[20].CommandType := DUT_CommandType.LogicCommand;
PersistentVars.Programs[10].Commands[20].CommandString := 'IF PASS THEN JUMP 24 ';
PersistentVars.Programs[10].Commands[20].CommandComment := 'jump over the counter operations';
PersistentVars.Programs[10].Commands[21].CommandType := DUT_CommandType.LogicCommand;
PersistentVars.Programs[10].Commands[21].CommandString := 'IF PASS THEN CNTRST 0 ';
PersistentVars.Programs[10].Commands[21].CommandComment := 'reset the column counter';
PersistentVars.Programs[10].Commands[22].CommandType := DUT_CommandType.LogicCommand;
PersistentVars.Programs[10].Commands[22].CommandString := 'IF PASS THEN CNTUP 1 ';
PersistentVars.Programs[10].Commands[22].CommandComment := 'increment the row counter';
PersistentVars.Programs[10].Commands[23].CommandType := DUT_CommandType.VarSetCommand;
PersistentVars.Programs[10].Commands[23].CommandString := 'STO 0 N 0.0 E 0.0 A 15.0 N 0.0 N 0.0 N 0.0 ';
PersistentVars.Programs[10].Commands[23].CommandComment := 'add the row width. clear column.';

//
FOR _i := GVL.PROG_CMDS_ARR_BEG TO GVL.PROG_CMDS_ARR_END BY 1 DO
	PersistentVars.Programs[15].Commands[_i].CommandType := DUT_CommandType.Disabled;
	PersistentVars.Programs[15].Commands[_i].CommandString := '';
	PersistentVars.Programs[15].Commands[_i].CommandComment := '';
END_FOR
PersistentVars.Programs[15].ProgramName := 'Gimbal 1';
PersistentVars.Programs[15].Commands[0].CommandType := DUT_CommandType.VarSetCommand;
PersistentVars.Programs[15].Commands[0].CommandString := 'STO 43 N 0.0 E 250.0 E 250.0 N 0.0 E 1.0e-2 E 1.0e-1 ';
PersistentVars.Programs[15].Commands[0].CommandComment := 'set velocity, acceleration, and jerk';
PersistentVars.Programs[15].Commands[1].CommandType := DUT_CommandType.VarSetCommand;
PersistentVars.Programs[15].Commands[1].CommandString := 'STO 43 E 100.0 E 1000.0 E 1000.0 E 1.0 E 1.0 E 1.0 ';
PersistentVars.Programs[15].Commands[1].CommandComment := 'set velocity, acceleration, and jerk';
PersistentVars.Programs[15].Commands[3].CommandType := DUT_CommandType.MoveCommand;
PersistentVars.Programs[15].Commands[3].CommandString := 'DIR ABS 30.0 ACS LIT -19.65 30.42 -55.18 0.0 4.04 0.0 ';
PersistentVars.Programs[15].Commands[3].CommandComment := 'Taught position';
PersistentVars.Programs[15].Commands[6].CommandType := DUT_CommandType.VarSetCommand;
PersistentVars.Programs[15].Commands[6].CommandString := 'STO 46 E 0.0 E 0.0 E 300.0 E 0.0 E 0.0 E 0.0 ';
PersistentVars.Programs[15].Commands[6].CommandComment := 'offset the TCP Z';
PersistentVars.Programs[15].Commands[7].CommandType := DUT_CommandType.MoveCommand;
PersistentVars.Programs[15].Commands[7].CommandString := 'LIN ABS 20.0 TCS LIT 0.0 0.0 0.0 0.0 -30.0 0.0 ';
PersistentVars.Programs[15].Commands[7].CommandComment := 'rotate around TCP Y';
PersistentVars.Programs[15].Commands[8].CommandType := DUT_CommandType.MoveCommand;
PersistentVars.Programs[15].Commands[8].CommandString := 'LIN ABS 20.0 TCS LIT 0.0 0.0 0.0 90.0 60.0 -90.0 ';
PersistentVars.Programs[15].Commands[8].CommandComment := 'rotate around TCP X with z$' y z$'$'';
PersistentVars.Programs[15].Commands[10].CommandType := DUT_CommandType.MoveCommand;
PersistentVars.Programs[15].Commands[10].CommandString := 'DIR ABS 30.0 ACS LIT -19.65 30.42 -55.18 0.0 4.04 0.0 ';
PersistentVars.Programs[15].Commands[10].CommandComment := 'Taught position';
PersistentVars.Programs[15].Commands[12].CommandType := DUT_CommandType.VarSetCommand;
PersistentVars.Programs[15].Commands[12].CommandString := 'STO 43 E 100.0 E 1000.0 E 1000.0 E 1.0 E 1.0 E 1.0 ';
PersistentVars.Programs[15].Commands[12].CommandComment := 'set velocity, acceleration, and jerk';
